FUNCTION F_LeakMonitor_LOTAO_1 : FB_LeakMonitor
VAR_INPUT
END_VAR
VAR_OUTPUT
	// Provide stBoundaries output so test functions can reuse the boundaries
	stBoundaries : ST_LeakBoundaries := F_LeakBoundaries();
END_VAR
VAR
	fbLeakMonitor : FB_LeakMonitor;
END_VAR

fbLeakMonitor(
	bLeakDetected := TRUE,
	bAmphosOn := TRUE,
	nLocationResistance := stBoundaries.nLMax4 - 1,
	stBound := stBoundaries
);

F_LeakMonitor_LOTAO_1 := fbLeakMonitor;

END_FUNCTION

(* stored: Version 1.1.0.1, ProductVersion 3.1.4024.0
   POU F_LeakMonitor_LOTAO_1: Id {7d02be5b-6272-4cb1-bc98-e349dc50b5f8}, SpecialFunc None *)
